{attribute addProperty BoxType "BK1150-0000-0018"}
{attribute addProperty Id "Term_385_KL1002KL1002_D229A9CA00"}
{attribute addProperty CRC "3685972702"}
{attribute addProperty SizeInBites "0"}
{attribute addProperty SizeInBytes "0"}
TYPE A_0012_BK1150_0000_0018_DBB37ADE EXTENDS BK1150_A5F67C82 :
STRUCT
	{attribute addProperty Name "Term_385_KL1002"}
	Term_385_KL1002 : KL1002_D229A9CA;
END_STRUCT
END_TYPE

(* stored: Version 1.2.0.0, ProductVersion 3.1.4024.9
   DUT A_0012_BK1150_0000_0018_DBB37ADE: Id {af9456c3-5938-4a4a-9ba9-d041f47e3364} *)
